FUNCTION_BLOCK XTSHardware EXTENDS CyclicBase IMPLEMENTS I_Initialisable, I_XtsHardware, I_Object
VAR
	XtsParts : ARRAY[0..TcIoXtsEnvironmentParameterList.MaxPartsPerTrack] OF XtsPart;
	IXtsParts : ARRAY[0..TcIoXtsEnvironmentParameterList.MaxPartsPerTrack] OF XtsPart;
	_MyNumberParts : INT;
	XtsTracks : ARRAY[0..TcIoXtsEnvironmentParameterList.MaxXtsTracksPerXpu] OF XtsTrack;
	IXtsTracks : ARRAY[0..TcIoXtsEnvironmentParameterList.MaxXtsTracksPerXpu] OF XtsTrack;
	_MyNumberTracks : INT;
	TrackOTCIDs: ARRAY [1..Tc3_XTS_Utility.TcIoXtsEnvironmentParameterList.MaxXtsTracksPerXpu] OF Tc3_XTS_Utility.OTCID;
	_MyXpu : Tc3_XTS_Utility.I_TcIoXtsProcessingUnit;
	XtsIoEnvInitialiseState : XtsHardwareInitialisation;
	MyPartCount: UDINT;
	MyTrackCount: UDINT;
	bMoverIdDetectionActive: BOOL;
	bMoverIdDetectionError: BOOL;
	bMoverIdDetected: BOOL;
	_MyXts : INT := 1;
	_MyName : STRING;
	_isInitialised: BOOL;
	_hasXPU : BOOL;
END_VAR

METHOD AreAllMoverPositionsValid : BOOL
VAR_INPUT
END_VAR
 IF _MyXpu.GetAreAllPositionsValid() THEN
	 AreAllMoverPositionsValid := TRUE;
 END_IF
END_METHOD

METHOD AreAnyPartsInError : BOOL
VAR
	i : INT;
END_VAR
FOR i := 0 TO TO_INT(MyPartCount - 1) DO
	IF XtsParts[i].HasError() THEN
		AreAnyPartsInError := TRUE;
	END_IF
END_FOR
END_METHOD

METHOD AreExpectedMoversFound : BOOL
VAR_INPUT
END_VAR
AreExpectedMoversFound := _MyXpu.GetExpectedMoverCount() = _MyXpu.GetDetectedMoverCount();
END_METHOD

METHOD PUBLIC  Cycle : HRESULT
VAR
	i : UDINT;
END_VAR
IF NOT _isInitialised THEN
	Cycle := -1;
	RETURN;
END_IF


FOR i := 0 TO (MyPartCount - 1) DO
	XtsParts[i].Cycle();
END_FOR
FOR i := 0 TO (MyTrackCount-1) DO
	XtsTracks[i].Cycle();
END_FOR
END_METHOD

PROPERTY DetectedNumberOfParts : INT
GET
DetectedNumberOfParts := TO_INT(_MyNumberParts);
END_GET
END_PROPERTY

PROPERTY DetectedNumberOfTracks : UINT
GET
DetectedNumberOfTracks := TO_UINT( MyTrackCount);
END_GET
END_PROPERTY

PROPERTY ExpectedNumberOfParts : int
GET
ExpectedNumberOfParts := _MyNumberParts;
END_GET
SET
_MyNumberParts := ExpectedNumberOfParts;
END_SET
END_PROPERTY

PROPERTY ExpectedNumberOfTracks : int
GET
ExpectedNumberOfTracks := _MyNumberTracks;
END_GET
SET
_MyNumberTracks := ExpectedNumberOfTracks;
END_SET
END_PROPERTY

METHOD GetConfiguredDetectionMoverNumber : UDINT
VAR_INPUT
END_VAR
GetConfiguredDetectionMoverNumber := _MyXpu.GetConfiguredDetectionCount();
END_METHOD

METHOD GetMoverDetectionState : DetectionStateEnum
VAR_INPUT
END_VAR
GetMoverDetectionState := _MyXpu.GetDetectionState();
END_METHOD

METHOD GetNumberMoversDetected : UDINT
VAR_INPUT
END_VAR
getNumberMoversDetected := _MyXpu.GetDetectedMoverCount();
END_METHOD

METHOD GetPartErrorCode : UDINT
VAR
	i : INT; 
	errorCode : UDINT;
END_VAR
FOR i := 0 TO TO_INT(MyPartCount - 1) DO
	IF XtsParts[i].GetCurrentError() <> 0 THEN
		errorCode := XtsParts[i].GetCurrentError();
		IF errorCode > GetPartErrorCode THEN
			GetPartErrorCode := errorCode;
		END_IF
	END_IF
END_FOR
END_METHOD

METHOD GetTrackInterfaceByNumber : I_XtsTrack
VAR_INPUT
	TrackNumber : UINT;
END_VAR
IF TrackNumber = 0 OR TrackNumber > MyTrackCount THEN
	GetTrackInterfaceByNumber := 0;
	RETURN;
END_IF
GetTrackInterfaceByNumber := XtsTracks[TrackNumber - 1];
END_METHOD

METHOD GetTrackInterfaceByOTCID : I_XtsTrack
VAR_INPUT
	trackOTCID : OTCID;
END_VAR
VAR
	i: INT;
END_VAR
FOR i := 0 TO _MyNumberTracks - 1 DO
	IF trackOTCID = XtsTracks[i].MyOTCID THEN
		GetTrackInterfaceByOTCID := XtsTracks[i];
	END_IF
END_FOR
END_METHOD

METHOD HasValidXPUReference : BOOL
VAR_INPUT
END_VAR
HasValidXPUReference := _hasXPU;
END_METHOD

METHOD Initialise : HRESULT
VAR
	i: INT;
	allInitialised : BOOL;
END_VAR
Initialise := -1;
CASE XtsIoEnvInitialiseState OF
	XtsHardwareInitialisation.WaitingForXpu:
		IF _MyXpu = 0 THEN
			RETURN;
		ELSE
			_MyName := _MyXpu.P_ObjectName;
			XtsIoEnvInitialiseState := XtsHardwareInitialisation.GettingParts;
		END_IF
	XtsHardwareInitialisation.GettingParts:
		MyPartCount := _MyXpu.P_PartCount;
		IF TO_INT(MyPartCount) = _MyNumberParts THEN
			FOR i := 0 TO (TO_INT(MyPartCount) - 1) DO
				XtsParts[i].MyXtsIoEnvInterface := _MyXpu.PartTcIo(TO_UINT(i + 1));
				IXtsParts[i] := XtsParts[i];
				IF THIS^.IsXtsInSim() THEN
					XtsParts[i].SetInSim();
				END_IF
			END_FOR
			XtsIoEnvInitialiseState := XtsHardwareInitialisation.GettingTracks;
		ELSE
			XtsIoEnvInitialiseState := XtsHardwareInitialisation.InitialisationFault;
		END_IF
	XtsHardwareInitialisation.GettingTracks:
		MyTrackCount := _MyXpu.P_TrackCount;
		_MyXpu.GetTrackOids();
		TrackOTCIDs := _MyXpu.P_TrackOids;
		IF TO_INT(MyTrackCount) = _MyNumberTracks THEN
			FOR i := 0 TO UDINT_TO_INT(MyTrackCount - 1) DO
				XtsTracks[i].MyXtsIoEnvInterface := _MyXpu.TrackTcIo(TO_UINT(i + 1));
				XtsTracks[i].MyOTCID := TrackOTCIDs[i + 1];
				IXtsTracks[i] := XtsTracks[i];
			END_FOR
			XtsIoEnvInitialiseState := XtsHardwareInitialisation.InitialisingXtsParts;
		ELSE
			XtsIoEnvInitialiseState := XtsHardwareInitialisation.InitialisationFault;
		END_IF
	XtsHardwareInitialisation.InitialisingXtsParts:
		allInitialised := TRUE;
		FOR i := 0 TO UDINT_TO_INT(MyPartCount - 1) DO
			IF FAILED(XtsParts[i].Initialise()) THEN
				allInitialised := FALSE;
			END_IF
		END_FOR
		IF allInitialised THEN
			XtsIoEnvInitialiseState := XtsHardwareInitialisation.InitialisingXtsTracks;
		END_IF
	XtsHardwareInitialisation.InitialisingXtsTracks:
		allInitialised := TRUE;
		FOR i := 0 TO UDINT_TO_INT(MyTrackCount - 1) DO
			IF FAILED(XtsTracks[i].Initialise()) THEN
				allInitialised := FALSE;
			END_IF
		END_FOR
		IF allInitialised THEN
			XtsIoEnvInitialiseState := XtsHardwareInitialisation.Initialised;
		END_IF
	XtsHardwareInitialisation.Initialised:
		_isInitialised := TRUE;
		Initialise := 0;
END_CASE
END_METHOD

METHOD IsHardware24VdcOK : HRESULT
VAR
	i : UDINT;
END_VAR
FOR i := 0 TO (_MyXpu.P_PartCount -1) DO
	IF NOT XtsParts[i].Is24VBusOK() THEN
		IsHardware24VdcOK := -1;
	END_IF
END_FOR
END_METHOD

METHOD IsHardware48VdcOK : HRESULT
VAR
	i : UDINT;
END_VAR
FOR i := 0 TO (_MyXpu.GetPartCount() - 1) DO
	IF NOT XtsParts[i].Is48VBusOK() THEN
		IsHardware48VdcOK := -1;
	END_IF
END_FOR
END_METHOD

METHOD IsIDDetectionStandard : BOOL
VAR_INPUT
END_VAR
IsIDDetectionStandard := _MyXpu.GetMoverIdDetectionMode() = MoverIdDetectionMode.Standard;
END_METHOD

METHOD IsInitialised : BOOL
VAR_INPUT
END_VAR
IsInitialised := _isInitialised;
END_METHOD

METHOD IsXtsInSim : BOOL
VAR_INPUT
END_VAR
IF  _MyXpu.GetOperationMode() = OperationMode.Simulation  THEN
	IsXtsInSim := TRUE;
END_IF
END_METHOD

PROPERTY MyName : string
GET
MyName := _MyName;
END_GET
END_PROPERTY

PROPERTY MyXpu : I_TcIoXtsProcessingUnit
GET
MyXpu := _MyXpu;
END_GET
SET
_MyXpu := MyXpu;
_hasXPU := TRUE;
END_SET
END_PROPERTY

PROPERTY MyXts : INT
GET
MyXts := _MyXts;
END_GET
SET
_MyXts := MyXts;
END_SET
END_PROPERTY

METHOD RegisterWithParent
VAR_INPUT
	Runner	: I_HostObjects;
END_VAR
Runner.RegisterCyclic(THIS^);
Runner.RegisterInitialisable(THIS^);
END_METHOD

METHOD RemoveATrackFromDetection : HRESULT
VAR_INPUT
	TrackToRemove : UINT;
END_VAR
IF TrackToRemove = 0 THEN
	RemoveATrackFromDetection := -1;
	RETURN;
END_IF
IF TrackToRemove > MyTrackCount THEN
	RemoveATrackFromDetection := -2;
	RETURN;
END_IF
IF MyTrackCount = 1 THEN
	RemoveATrackFromDetection := -3;
	RETURN;
END_IF
XtsTracks[TrackToRemove - 1].RemoveFromDetection();
END_METHOD

METHOD ResetAllParts : BOOL
VAR
	i : INT;
END_VAR
FOR i := 0 TO TO_INT(MyPartCount - 1) DO
	XtsParts[i].ResetPart();
	XtsParts[i].ResetNct();
END_FOR
END_METHOD

METHOD ResetAPart : HRESULT
VAR_INPUT
	Part : UINT;
END_VAR
IF Part > MyPartCount THEN
	ResetAPart := -1;
END_IF

IF Part = 0 THEN
	ResetAPart := -2;
END_IF

XtsParts[Part].ResetPart();
XtsParts[Part].ResetNct();
END_METHOD

METHOD SetAPartOriginTransform : BOOL
VAR_INPUT
	Part : INT;
	OriginTransform: Tc3_XTS_Utility.ST_OriginTransform;
END_VAR
XtsParts[Part - 1].SetPartOriginTransform(OriginTransform);
END_METHOD

METHOD SetATrackForDetection : HRESULT
VAR_INPUT
	TrackToDetect : UINT;
END_VAR
IF TrackToDetect = 0 THEN
	SetATrackForDetection := -1;
	RETURN;
END_IF
IF TrackToDetect > MyTrackCount THEN
	SetATrackForDetection := -2;
	RETURN;
END_IF

XtsTracks[TrackToDetect - 1].SetForDetection();
END_METHOD

METHOD SetMoverNumberForDetection : HRESULT
VAR_INPUT
	NumberOfMovers : INT;
END_VAR
IF NumberOfMovers < 0 THEN
	SetMoverNumberForDetection := -1;
	RETURN;
END_IF
IF NumberOfMovers > _MyXpu.GetMoverCount() THEN
	SetMoverNumberForDetection := -2;
	RETURN;
END_IF
 
_MyXpu.SetConfiguredDetectionCount(nConfiguredMoverDetectionCount := TO_UDINT(NumberOfMovers));
END_METHOD

METHOD TriggerMoverDetection : HRESULT
VAR_INPUT
END_VAR
IF _MyXpu = 0 THEN
	TriggerMoverDetection := -1;
	RETURN;
END_IF
_MyXpu.TriggerDetection();
END_METHOD

METHOD TriggerMoverIDDetection : HRESULT
VAR_INPUT
END_VAR
bMoverIdDetectionError 	:= _MyXpu.GetHasMoverIdDetectionError();
bMoverIdDetected 	:= _MyXpu.GetIsMoverIdDetectionValid();
bMoverIdDetectionActive	:= _MyXpu.GetIsMoverIdDetectionActive();

IF _MyXpu.GetMoverIdDetectionMode() = MoverIdDetectionMode.Standard THEN
	TriggerMoverIDDetection := -1;
	RETURN;
END_IF
// 
IF bMoverIdDetectionActive THEN
	TriggerMoverIDDetection := -2;
	RETURN;
END_IF

_MyXpu.TriggerMoverIdDetection();
END_METHOD

METHOD TriggerMoverRedetection : HRESULT
VAR_INPUT
END_VAR
IF _MyXpu = 0 THEN
	TriggerMoverRedetection := -1;
	RETURN;
END_IF

_MyXpu.TriggerRedetection();
END_METHOD

END_FUNCTION_BLOCK

(* stored: Version 1.1.0.1
   POU XTSHardware: Id {2082c175-1a19-4a3f-b920-8dbd46477756}, SpecialFunc None
   Folder Commands: Id {fac9eba9-c7de-4a76-a05e-49072f1b1bf8}
   Folder Settings: Id {977db0ee-8b4c-4e4e-adde-487140886b9b}
   Folder Status: Id {1e7de418-5187-4871-82b8-ce216901bd03}
   Method AreAllMoverPositionsValid: Id {61902ec7-4049-4544-9a8e-27dabf1b61be}
   Method AreAnyPartsInError: Id {699ab4e2-69ca-4162-ab63-9b7de63fc2c4}
   Method AreExpectedMoversFound: Id {642f39f7-45fb-4e7e-95d2-cca7f46c73a6}
   Method Cycle: Id {907368a2-7640-4dfa-a8a9-6f1d20861921}
   Property DetectedNumberOfParts: Id {0cb9ae9e-f39b-4029-894a-e6620c4ecf6f}
   Get Get: Id {c6657b2f-e5c5-4f83-9cec-2457aaa61cb5}
   Property DetectedNumberOfTracks: Id {1aee3abf-438c-401a-96dd-e5d65d11e759}
   Get Get: Id {6b1c17e2-83ee-47f8-b12c-999752617527}
   Property ExpectedNumberOfParts: Id {a98ec162-431e-48cc-ae6d-f8949630ea06}
   Get Get: Id {6aea69f8-39b7-432c-a6be-0e19820e9502}
   Set Set: Id {3a096234-62c8-4cae-b087-998329491864}
   Property ExpectedNumberOfTracks: Id {4b737a8f-2e1c-463e-a095-5f8b64b3f222}
   Get Get: Id {42884cba-9387-4d1f-8822-97815c1c289f}
   Set Set: Id {615cc55c-cb9a-4994-a6a7-0d139d5ef074}
   Method GetConfiguredDetectionMoverNumber: Id {43f766d9-966d-4623-a223-676c73e2281d}
   Method GetMoverDetectionState: Id {5c04b4df-babc-44c4-8315-87ac6e89bad7}
   Method GetNumberMoversDetected: Id {6134912a-11cc-419f-9366-ca4c2c2c2f9f}
   Method GetPartErrorCode: Id {1db9bad9-9f3a-4db0-b023-7e6033e80429}
   Method GetTrackInterfaceByNumber: Id {f2581b5d-dcdf-4c20-8ad6-39f08544aef0}
   Method GetTrackInterfaceByOTCID: Id {d55b1037-e87a-4176-a531-719c46a289ea}
   Method HasValidXPUReference: Id {6ea3239f-d8a6-4ea4-a8cf-a5b51d9c01b2}
   Method Initialise: Id {95822be7-e433-46ff-bfc3-e4b3c51e2a74}
   Method IsHardware24VdcOK: Id {16c30a69-c544-4706-ba78-c8aed5346201}
   Method IsHardware48VdcOK: Id {ff4a117c-24f4-4466-b159-c15d29dc7330}
   Method IsIDDetectionStandard: Id {aa7a18ac-0236-4a73-a20e-a9a08158b988}
   Method IsInitialised: Id {550c07cc-fb09-419f-9cfc-c551f12c3cb9}
   Method IsXtsInSim: Id {c26b05e6-e2eb-40cc-bea5-adcd4dafa0e7}
   Property MyName: Id {0d9f86cc-11b2-415a-83b4-e3fe22742bf6}
   Get Get: Id {05735f6c-e3fe-4ee3-a217-5178eba283c4}
   Property MyXpu: Id {9f0e6f27-b8f0-452c-b07d-d4d2a7ed1b3b}
   Get Get: Id {ef18a883-259a-46c5-ac1a-fd1d0138159b}
   Set Set: Id {3f18a9fd-c75b-45a9-b0a5-a4cb82b21b6b}
   Property MyXts: Id {97cba7e2-9698-4397-a6b4-6da9e2abe688}
   Get Get: Id {ad7d6d73-4fab-4d05-975f-01e196f73334}
   Set Set: Id {7ade4ba5-90b5-400a-aadf-8d737611d6d9}
   Method RegisterWithParent: Id {cc909a39-cbe3-4035-b5c9-fc3340c04e55}
   Method RemoveATrackFromDetection: Id {1e31681d-3ada-48de-80fd-ab8c9694949c}
   Method ResetAllParts: Id {62a3421b-7f58-4518-b99a-efef3044ec5b}
   Method ResetAPart: Id {917224af-ad90-4e18-bee4-fe5c99cd4d59}
   Method SetAPartOriginTransform: Id {603deaa6-bf5d-4b68-a30f-e30620f70274}
   Method SetATrackForDetection: Id {33a6fd5d-a8a8-4e54-be38-eeae850dd3e9}
   Method SetMoverNumberForDetection: Id {fda2cbfb-05d3-433d-b308-26404cfa0e4a}
   Method TriggerMoverDetection: Id {15e78533-ebfe-46e6-bd25-18e4044d6883}
   Method TriggerMoverIDDetection: Id {23436421-ecb3-466c-b86b-5fefe5c7904c}
   Method TriggerMoverRedetection: Id {0183a3e0-45ff-4ec4-b868-d12cfe75fb77} *)
